{attribute 'linkalways'} 
{attribute 'no_explicit_call' := 'This FB is a CLASS and must be accessed using methods or properties'}
{attribute 'enable_dynamic_creation'}
FUNCTION_BLOCK Node_F_VN_MinElementElementwise_UDINT EXTENDS VisionNode
VAR
    ipContainer : _ITcVnContainer;
    nMin : _UDINT(0);
    hrPrev : _HRESULT(S_OK);
    hresult : _HRESULT(S_OK);
END_VAR

METHOD PUBLIC  Clone : I_Node
VAR
	pNode : POINTER TO Node_F_VN_MinElementElementwise_UDINT;
END_VAR
pNode := __NEW(Node_F_VN_MinElementElementwise_UDINT);
Clone := pNode^;
END_METHOD

METHOD FB_init : BOOL
VAR_INPUT
	bInitRetains : BOOL; // if TRUE, the retain variables are initialized (warm start / cold start)
	bInCopyCode : BOOL;  // if TRUE, the instance afterwards gets moved into the copy code (online change)
END_VAR
AddInput('ipContainer', ipContainer);
AddInput('hrPrev', hrPrev);
AddOutput('ipContainer', ipContainer);
AddOutput('nMin', nMin);
AddOutput('hresult',hresult);
END_METHOD

METHOD PROTECTED OnExecute
hresult.Value := F_VN_MinElementElementwise_UDINT(
    ipContainer := ipContainer.Value,
    nMin := nMin.Value,
    hrPrev:= hrPrev.Value);
END_METHOD

METHOD PUBLIC PreExecutionCheck
VAR_INPUT
	Check : I_PreExecutionChecks;
END_VAR
Check.IsTrue(ipContainer.IsValid, 'ipContainer must be a valid container');
Check.IsTrue(ipContainer.IsType(TC_GLOBAL_CONST_LIST.ContainerType_Vector_UDINT), 'ipContainer contains incorrect type');
END_METHOD

END_FUNCTION_BLOCK

(* stored: Version 1.1.0.1, ProductVersion 3.1.4026.13
   POU Node_F_VN_MinElementElementwise_UDINT: Id {1deb9d36-325b-4258-a37f-fccad72b1e0d}, SpecialFunc None
   Folder Constructor: Id {ee930236-9694-476c-b216-6d252aa967e7}
   Method Clone: Id {daa12744-c21a-4b71-85bc-1cd85514472c}
   Method FB_init: Id {aa4ce294-a951-4677-ab3a-2710c774496b}
   Method OnExecute: Id {66ee562c-a4d2-4a56-aab1-ec1b0f764706}
   Method PreExecutionCheck: Id {8f791647-9a3b-4cc7-9812-35474e3d76d9} *)
